// TIA Portal V16 export
// export: Created 2023-01-04T15:44:09.7897286Z, ExportSetting WithDefaults, DisplayName Totally Integrated Automation Portal, DisplayVersion V16, DisplayName TIA Portal Version Control Interface, DisplayVersion V16, DisplayName TIA Portal Openness, DisplayVersion V16, DisplayName STEP 7 Professional, DisplayVersion V16, DisplayName STEP 7 Safety, DisplayVersion V16, DisplayName WinCC Advanced, DisplayVersion V16
DATA_BLOCK "DuplicateDB"   // DB12
{ S7_Optimized_Access := 'FALSE' }
VERSION : 0.1
// stored: AutoNumber true, DBAccessibleFromOPCUA true, IsOnlyStoredInLoadMemory false, IsWriteProtectedInAS false
   VAR
      Input : Struct
         FIC_B102 : Int;   // Tank2 Level Measurement
         LIC_B101 : Int;
         PS1_RFID_Station : Bool;
         PS2_Filling_Station : Bool;
         PS3_Quality_Station : Bool;
         PS4_End_of_Conveyor : Bool;
         T01_Low_Level : Bool;
         T01_High_Level : Bool;
      END_STRUCT;
   END_VAR
BEGIN
END_DATA_BLOCK
